// TIA Portal V17 export
// export: Created 2025-06-26T07:49:47.8554584Z, ExportSetting WithDefaults, DisplayName Totally Integrated Automation Portal, DisplayVersion V17 Update 8, DisplayName TIA Portal Openness, DisplayVersion V17 Update 8, DisplayName TIA Portal Version Control Interface, DisplayVersion V17, DisplayName STEP 7 Professional, DisplayVersion V17 Update 8, DisplayName STEP 7 Safety, DisplayVersion V17 Update 6, DisplayName WinCC Advanced, DisplayVersion V17 Update 8
FUNCTION_BLOCK "fbOneShot"   // FB56, FBD
TITLE = One-shot with trigger delay
{ S7_Optimized_Access := 'TRUE' }
AUTHOR : Heaten
VERSION : 0.1
// stored: AutoNumber true, IsIECCheckEnabled false, IsRetainMemResEnabled false, MemoryReserve 0, SetENOAutomatically false, UDAEnableTagReadback false
   VAR_INPUT
      bEnable : Bool;   // 1 = enable controller, 0 = disable
      tOnTime : Time;
      tStartDelay : Time;
   END_VAR
   VAR_OUTPUT
      bOut : Bool;
      tOnTimeElapsed : Time;
      tStartDelayElapsed : Time;
   END_VAR
   VAR
      StartDelayTimer : TON_TIME;
      OnTimer { S7_SetPoint := 'True'} : TP_TIME;
   END_VAR
BEGIN

REGION Network 1: Trigger delay
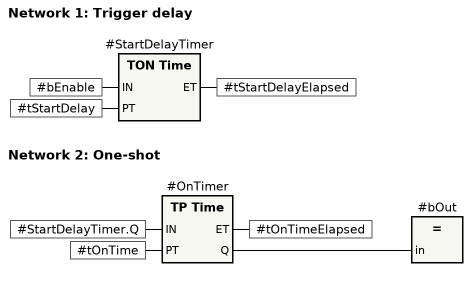
   #StartDelayTimer(IN := #bEnable, PT := #tStartDelay, ET => #tStartDelayElapsed);   // TON
END_REGION

REGION Network 2: One-shot
   #OnTimer(IN := #StartDelayTimer.Q, PT := #tOnTime, ET => #tOnTimeElapsed);   // TP
   #bOut := #OnTimer.Q;
END_REGION
END_FUNCTION_BLOCK
